(* IEC 61131-3 sources: CODESYS-IO-Visualization/CODESYS-IO-Visualization.fbsproj/Pi.device.xml.v3^/Plc Logic.plclogic.xml.v3^/Application.application.xml.v3^/Programs/2_Instruments, 1 file *)

(* ---- Main_Instruments.prg.st ---- *)
PROGRAM Main_Instruments
VAR
END_VAR

// Ambient Temperature: Site.Plant.AmbientTemp
InstA(Data := Site.Plant.AmbientTemp);

// Pump 1 Flow: Site.Plant.Pump1.Flow
InstA(Data := Site.Plant.Pump1.Flow);

// Pump 1 Temperature: Site.Plant.Pump1.Temp
InstA(Data := Site.Plant.Pump1.Temp);
